// TIA Portal V20 export
TYPE "LER_typePowerMC"
// stored: Access Published, IsFailsafeCompliant true, Namespace Safety
   STRUCT
      controlPowerFeedBack : Bool;
      controlPowerFeedBackVS : Bool;
      controlPowerOn : Bool;
      error : Bool;
      ackReq : Bool;
   END_STRUCT;
END_TYPE
